(* IEC 61131-3 sources: volt/packages/volt-lsp-iec/test-corpus/lenze-mid/Device/Plc Logic/Application/Library Manager/CAA ResMan, 24 files *)

(* ---- CLASS_INFO.dut ---- *)
TYPE CLASS_INFO :
STRUCT
	PFUNCTION : CAA.PVOID;
	CTMAXHANDLES : CAA.COUNT;
	CTACTHANDLES : CAA.COUNT;
END_STRUCT
END_TYPE

(* ---- ERROR.dut ---- *)
TYPE ERROR :
(
	NO_ERROR,
	FIRST_ERROR := 30300,
	HANDLE_INVALID := 30302,
	UNKNOWN_EVENT := 30303,
	NOMORE_MEMORY := 30304,
	PARAM_ERROR := 30305,
	WRONGOP_ERROR := 30306,
	GEN_ERROR := 30307,
	NOT_EMPTY := 30308,
	UNREGISTER_ERROR := 30309,
	REGISTER_ERROR := 30310,
	PARENT_OCCUPIED := 30311,
	CLASS_EMPTY := 30312,
	CLASS_FREE_ERROR := 30313,
	FIRST_MF := 30350,
	LAST_ERROR := 30399
);
END_TYPE

(* ---- INFO.dut ---- *)
TYPE INFO :
STRUCT
	CTMAXCOUNTCLASSES : CAA.COUNT;
	CTACTCOUNTCLASSES : CAA.COUNT;
END_STRUCT
END_TYPE

(* ---- RSM_HANDLE.dut ---- *)
TYPE RSM_HANDLE :
STRUCT
	PNEXT : CAA.PVOID;
	PPREV : CAA.PVOID;
	HHANDLE : CAA.HANDLE;
END_STRUCT
END_TYPE

(* ---- VERSIONCONSTANTS.gvl ---- *)
VAR_GLOBAL
	GC_BYVERSION : BYTE := 1;
	GC_BYVERSION_1 : BYTE := 0;
END_VAR

(* ---- _BLOCKGETDATA.pou ---- *)
FUNCTION _BLOCKGETDATA : CAA.PVOID
VAR_INPUT
	HBLOCK : CAA.HANDLE;
	PEERROR : POINTER TO ERROR;
END_VAR
END_FUNCTION

(* ---- _POOLCREATEP.pou ---- *)
FUNCTION _POOLCREATEP : CAA.HANDLE
VAR_INPUT
	SZBLOCKSIZE : CAA.SIZE;
	SZMEMSIZE : CAA.SIZE;
	PMEMORY : CAA.PVOID;
	EEMPTY : INT;
	PEERROR : POINTER TO ERROR;
END_VAR
END_FUNCTION

(* ---- _POOLDELETE.pou ---- *)
FUNCTION _POOLDELETE : ERROR
VAR_INPUT
	HPOOL : CAA.HANDLE;
END_VAR
END_FUNCTION

(* ---- _POOLEXTENDH.pou ---- *)
FUNCTION _POOLEXTENDH : ERROR
VAR_INPUT
	HPOOL : CAA.HANDLE;
	CTNUMBLOCKS : CAA.COUNT;
END_VAR
END_FUNCTION

(* ---- _POOLGETBLOCK.pou ---- *)
FUNCTION _POOLGETBLOCK : CAA.HANDLE
VAR_INPUT
	HPOOL : CAA.HANDLE;
	PEERROR : POINTER TO ERROR;
END_VAR
END_FUNCTION

(* ---- _POOLPUTBLOCK.pou ---- *)
FUNCTION _POOLPUTBLOCK : ERROR
VAR_INPUT
	HBLOCK : CAA.HANDLE;
END_VAR
END_FUNCTION

(* ---- CHECK.pou ---- *)
FUNCTION CHECK : CAA.HANDLE
VAR_INPUT
	HCHECK : CAA.HANDLE;
	PEERROR : POINTER TO ERROR;
END_VAR
END_FUNCTION

(* ---- CLASSCREATE.pou ---- *)
FUNCTION CLASSCREATE : CAA.HANDLE
VAR_INPUT
	PFUNCTION : CAA.PVOID;
	CTMAXHANDLES : CAA.COUNT;
	PEERROR : POINTER TO ERROR;
END_VAR
END_FUNCTION

(* ---- CLASSDELETE.pou ---- *)
FUNCTION CLASSDELETE : ERROR
VAR_INPUT
	HCLASS : CAA.HANDLE;
END_VAR
END_FUNCTION

(* ---- CLASSFREE.pou ---- *)
FUNCTION CLASSFREE : ERROR
VAR_INPUT
	HCLASS : CAA.HANDLE;
END_VAR
END_FUNCTION

(* ---- GETCLASS.pou ---- *)
FUNCTION GETCLASS : CAA.HANDLE
VAR_INPUT
	HCHECK : CAA.HANDLE;
	PEERROR : POINTER TO ERROR;
END_VAR
END_FUNCTION

(* ---- GETCLASSINFO.pou ---- *)
FUNCTION GETCLASSINFO : ERROR
VAR_INPUT
	HCLASS : CAA.HANDLE;
	PCLASSINFO : POINTER TO CLASS_INFO;
END_VAR
END_FUNCTION

(* ---- GETINFO.pou ---- *)
FUNCTION GETINFO : ERROR
VAR_INPUT
	PINFO : POINTER TO INFO;
END_VAR
END_FUNCTION

(* ---- GETPARENT.pou ---- *)
FUNCTION GETPARENT : CAA.HANDLE
VAR_INPUT
	HCHECK : CAA.HANDLE;
	PEERROR : POINTER TO ERROR;
END_VAR
END_FUNCTION

(* ---- GETSUPPLIERVERSION.pou ---- *)
FUNCTION GETSUPPLIERVERSION : WORD
VAR_INPUT
	XDUMMY : BOOL;
END_VAR
END_FUNCTION

(* ---- REGISTER.pou ---- *)
FUNCTION REGISTER : CAA.HANDLE
VAR_INPUT
	HCLASS : CAA.HANDLE;
	HRESSOURCE : CAA.HANDLE;
	PEERROR : POINTER TO ERROR;
END_VAR
END_FUNCTION

(* ---- SETPARENT.pou ---- *)
FUNCTION SETPARENT : ERROR
VAR_INPUT
	HCHECK : CAA.HANDLE;
	HCHECKPARENT : CAA.HANDLE;
END_VAR
END_FUNCTION

(* ---- UNREGISTER.pou ---- *)
FUNCTION UNREGISTER : ERROR
VAR_INPUT
	HCHECK : CAA.HANDLE;
END_VAR
END_FUNCTION

(* ---- RSMCLASS.pou ---- *)
FUNCTION_BLOCK RSMCLASS
VAR
	_HPOOL : CAA.HANDLE;
	_ADWPOOL : ARRAY [0..19] OF __XWORD;
	_PLIST : POINTER TO RSM_HANDLE;
END_VAR
END_FUNCTION_BLOCK

METHOD FB_EXIT : BOOL
VAR_INPUT
	BINCOPYCODE : BOOL;
END_VAR
END_METHOD

METHOD REGISTER : CAA.HANDLE
VAR_INPUT
	HHANDLE : CAA.HANDLE;
	PEERROR : POINTER TO ERROR;
END_VAR
END_METHOD

METHOD CLOSE : ERROR
VAR_INPUT
	HHANDLE : CAA.HANDLE;
END_VAR
END_METHOD

METHOD SEARCH : CAA.HANDLE
VAR_INPUT
	HHANDLE : CAA.HANDLE;
END_VAR
END_METHOD

METHOD UNREGISTER : ERROR
VAR_INPUT
	HHANDLE : CAA.HANDLE;
END_VAR
END_METHOD

METHOD FB_INIT : BOOL
VAR_INPUT
	BINITRETAINS : BOOL;
	BINCOPYCODE : BOOL;
END_VAR
END_METHOD

METHOD TRANSLATE : CAA.HANDLE
VAR_INPUT
	HHANDLE : CAA.HANDLE;
END_VAR
VAR_OUTPUT
	EERROR : ERROR;
END_VAR
END_METHOD
